PROGRAM P_MachineLog
VAR
	
	fbFilePuts: FB_FilePuts;
	fbFileClose: FB_FileClose;
	fbFileOpen: FB_FileOpen;
	iStep :INT;
	bFileOpened		:BOOL;
	sFileName		:STRING;
	hHandle			:UINT;	
	i				:INT; 
END_VAR

CASE iStep OF
	0:
		IF	GVL_General.LogBufferIndex >0 THEN 
			iStep := 10;
		ELSIF bFileOpened=TRUE THEN 
			iStep := 50;			
		END_IF
	10: (* check the file is open or not*)
		IF NOT bFileOpened THEN 
			iStep := 11;
		ELSE
			iStep := 20; 
		END_IF
	11:		(* try to open the file*)
		sFileName := CONCAT(STR1:= GVL_General.sFilePath,STR2:= F_DateNow());
		sFileName := CONCAT(STR1:= sFileName,'.txt');
		fbFileOpen(sNetId:= ,sPathName:= ,nMode:= ,ePath:= ,bExecute:= FALSE ,
					tTimeout:=T#3S ,bBusy=> ,bError=> ,nErrId=> ,hFile=> );
		IF NOT	fbFileOpen.bBusy AND NOT fbFileOpen.bError THEN 
			iStep := 12;
		END_IF
	12:	(* open the file or create the file*)
		
		fbFileOpen(sNetId:= ,sPathName:= sFileName,nMode:= FOPEN_MODEAPPEND ,ePath:= PATH_GENERIC ,bExecute:= TRUE ,
					tTimeout:=T#3S ,bBusy=> ,bError=> ,nErrId=> ,hFile=> hHandle);
		IF NOT fbFileOpen.bBusy AND NOT fbFileOpen.bError THEN 
			bFileOpened := TRUE;
			iStep := 20;
		END_IF
		
	20: (* try to write to the log file*)
		fbFilePuts(sNetId:= ,hFile:=hHandle ,sLine:=, bExecute:=FALSE,tTimeout:=T#3S,bBusy=> ,bError=> ,nErrId=> );
		IF NOT fbFilePuts.bBusy AND NOT fbFilePuts.bError THEN 
			iStep := 21;
		END_IF
	21:
		fbFilePuts(sNetId:= ,hFile:=hHandle ,sLine:=GVL_General.LogBufferArray[1],bExecute:=TRUE,tTimeout:=T#3S,bBusy=> ,bError=> ,nErrId=> );
		IF	NOT fbFilePuts.bBusy AND NOT fbFilePuts.bError THEN 
			//GVL_General.LogBufferIndex := GVL_General.LogBufferIndex -1;		//???
			iStep := 22;
		END_IF
	22:
		
			FOR i := 1 TO GVL_General.LogBufferIndex - 1 DO
				GVL_General.LogBufferArray[i] := GVL_General.LogBufferArray[i + 1];
			END_FOR
			GVL_General.LogBufferIndex := GVL_General.LogBufferIndex -1;		//???
		IF	GVL_General.LogBufferIndex >1 THEN 
			
			iStep := 0;
		ELSE 
			iStep := 50;
		END_IF
	
	50:
		fbFileClose(sNetId:= ,hFile:= fbFileOpen.hFile,bExecute:=FALSE,tTimeout:=T#3S ,	bBusy=> ,bError=> ,nErrId=> );
		IF NOT fbFileClose.bBusy THEN 
			IF NOT fbFileClose.bError THEN 
				iStep:= 51;
			END_IF
		END_IF
		
	51:
		fbFileClose(sNetId:= ,hFile:=fbFileOpen.hFile,bExecute:=TRUE,tTimeout:=T#3S,bBusy=> ,bError=> ,nErrId=> );
		
		IF NOT fbFileClose.bBusy THEN 
			IF NOT fbFileClose.bError THEN
				bFileOpened := FALSE;
				iStep := 0;
			ELSE 
				iStep := 999;
			END_IF
		END_IF
	999:
		;
END_CASE

END_PROGRAM

(* stored: Version 1.1.0.1, ProductVersion 3.1.4022.16
   POU P_MachineLog: Id {6c67e9a0-f750-4f40-a501-684ac4c18bfd}, SpecialFunc None *)
